KUKA KRL program: WL_TASMOCIAG.src

&ACCESS RVP
&REL 1
&PARAM TEMPLATE = C:\KRC\Roboter\Template\ExpertVorgabe
&PARAM EDITMASK = *
DEF WL_TASMOCIAG(CZY_WLACZYC :IN)

BOOL CZY_WLACZYC

IF CZY_WLACZYC == TRUE THEN
TASMOCIAG_KROKOWO(-1,3)
ELSE
TASMOCIAG_KROKOWO(0,0)
ENDIF

END
